Staubli VAL3: ChangeCpoint.pgx

public program ChangeCpoint(trsf& x_trSource[], num x_nDia, bool& x_bRes)
  local trsf l_trTrsf
  local num l_nDia
  local num l_nNum
begin
  //根据直径来修改点的数值
  //外接圆

  //先根据三点来获得圆心点，然后根据三个点来求的圆心与三个点的长度。



  x_bRes=false

  if size(x_trSource)!=3
    return
  endIf


  call Circumcircle(x_trSource,l_trTrsf,l_nDia,x_bRes)
  if !x_bRes
    return
  endIf

  for l_nNum=0 to 2
    call ChangeCirPoint(l_trTrsf,x_nDia,x_trSource[l_nNum],x_trSource[sel(l_nNum==2,0,l_nNum+1)],x_bRes)
    if !x_bRes
      return
    endIf
  endFor

end
